Universal Robots PolyScope program: robotiq_gripper_python.urp

Program robotiq_gripper_python (installation=robotiq_gripper_python directory=/programs/usbdisk/CPS_MUL createdIn=5.15.2 lastSavedIn=5.15.2 robotSerialNumber=20225300304)
Calibrated DH parameters: a=[-0.000098, -0.243076, -0.21071, 0.00009, -0.000141, 0]; d=[0.151916, 6.117956, 1.286418, -7.27361, 0.085314, 0.092309]; alpha=[1.571347, -0.002639, 0.004542, 1.571514, -1.572056, 0]; deltaTheta=[0, -0.066307, 0.224581, -0.158277, 0.000001, 0]
InitVariablesNode
Robot Program (runOnlyOnce=false)
  URCap Gripper (Robotiq_Grippers, Robotiq Inc.) dataModel(position=1.1764705882352942, force=60.0, speed=60.0, positionInDouble=1.1764705882352942, forceInDouble=60.0, speedInDouble=60.0, slaveIds=[9], blocking=true)
  Loop Forever
    Wait Sleep waitTime=0.1
